FUNCTION_BLOCK FB_GetCPULoad
VAR_INPUT
	rInterval			: REAL := 10.0;		// [sec]
END_VAR
VAR_OUTPUT
	rCPULoad			: REAL;				// [%]
	rCPUFrequency		: REAL;
	bError				: BOOL;				// error flag (indicator: error occured)
	nErrID				: UDINT;			// last error ID 
END_VAR
VAR
	// internal use
	sAmsNetId			: STRING := '';		// ADS Net ID (local = '')    
	iState				: INT;
	uData				: UINT;
    stMDP_ModuleHeader  : ST_MDP_ModuleHeader;
    stMDP_ModuleContent : ST_MDP_CPU;
	// FB instances
	fbReadMDPCPU		: Tc2_MDP.FB_MDP_CPU_Read;
	tonInterval			: Tc2_Standard.TON;
	// Info
	iErrorCnt			: UINT;
	iGoodCnt			: UINT;
END_VAR


// Interval timer
tonInterval(IN := NOT tonInterval.Q, PT := REAL_TO_TIME(rInterval * 1000.0));

CASE iState OF
	0: // Initiate program parameters (if required)
		fbReadMDPCPU(bExecute := FALSE);
		IF (tonInterval.Q) THEN
			iState := 10;
		END_IF

	10:	// Trigger FB: request CPU data
		fbReadMDPCPU(	bExecute := TRUE,
						tTimeout := T#5S,
						iModIdx := 0,
						sAmsNetId := sAmsNetId,
						stMDP_ModuleHeader => stMDP_ModuleHeader,
						stMDP_ModuleContent => stMDP_ModuleContent 	);
		iState := 20;

	20:	// Process FB: Request CPU temp
		fbReadMDPCPU(bExecute := FALSE); 
		IF (NOT fbReadMDPCPU.bBusy) THEN
			IF (fbReadMDPCPU.bError) THEN
				bError := TRUE;
				nErrID := fbReadMDPCPU.nErrID; 
				iErrorCnt := iErrorCnt + 1;
				iState := 0;
			ELSE
				bError := FALSE;
				rCPULoad := UINT_TO_REAL(stMDP_ModuleContent.iCPUusage);
				rCPUFrequency := UDINT_TO_REAL(stMDP_ModuleContent.iCPUfrequency);
				iGoodCnt := iGoodCnt + 1;
				iState := 30;
			END_IF                                               
		END_IF
    
     30: // Done 
		iState := 0;

	ELSE
		iState := 0; 

END_CASE

END_FUNCTION_BLOCK

(* stored: Version 1.1.0.1, ProductVersion 3.1.4024.5
   POU FB_GetCPULoad: Id {70ee7357-34f0-4162-9fda-b8bdd33a860a}, SpecialFunc None *)
